// Mitsubishi GX Works2 project: FinalProject   PLC: FX3U/FX3UC

// global labels: Global1
VAR_GLOBAL
  Pos_RedArea AT D109 : INT;
  Pos_AreaA AT D110 : INT;
  End_Home AT M300 : BOOL;
  End_Prepare AT M301 : BOOL;
  Move_Home AT M329 : BOOL;
  En_GetA AT M303 : BOOL;
  GetA AT M304 : BOOL;
  En_GoRed AT M305 : BOOL;
  Go_Red AT M306 : BOOL;
  En_GoBlue AT M307 : BOOL;
  GoBlue AT M308 : BOOL;
  En_Go_A AT M309 : BOOL;
  Go_A AT M310 : BOOL;
  En_Go_B AT M311 : BOOL;
  Go_B AT M312 : BOOL;
  En_GetB AT M313 : BOOL;
  GetB AT M314 : BOOL;
  M_Dem AT M315 : BOOL;
  End_Arr_Red AT M317 : BOOL;
  M_timer AT M318 : BOOL;
  Start_Home AT M319 : BOOL;
  End_ComeBack AT M320 : BOOL;
  Start_B AT X003 : BOOL;
  Stop_B AT X004 : BOOL;
  Emer_B AT M323 : BOOL;
  Go_Home AT M324 : BOOL;
  END_GOHOME AT M325 : BOOL;
  end_get_ProA AT M326 : BOOL;
  M_Xoay AT M327 : BOOL;
  End_RedArea AT M328 : BOOL;
  M_T1 AT M330 : BOOL;
  M_Arr AT M331 : BOOL;
  M_T2 AT M332 : BOOL;
  M_T3 AT M333 : BOOL;
  M_T7 AT M334 : BOOL;
  M_ComeBack AT M335 : BOOL;
  End_Finish AT M336 : BOOL;
  M_T5 AT M337 : BOOL;
  M_Prepare AT S338 : BOOL;
  M_Start AT M321 : BOOL;
  M_Stop AT M322 : BOOL;
END_VAR

PROGRAM MAIN
VAR
  Move_Data_1 : Move_Data;
END_VAR
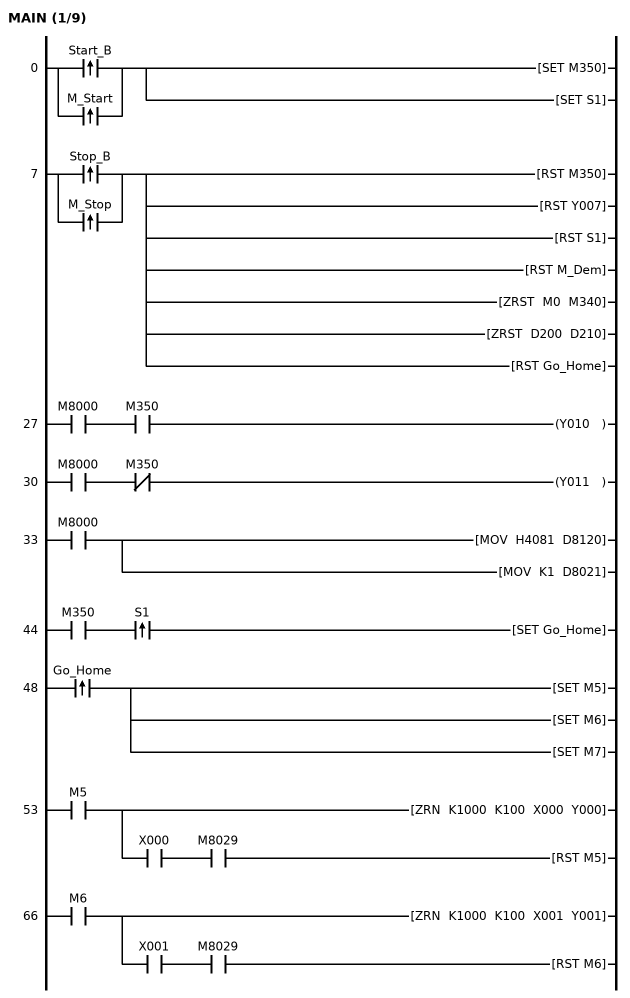
0     LDP     Start_B
      ORP     M_Start
      SET     M350
      SET     S1
7     LDP     Stop_B
      ORP     M_Stop
      RST     M350
      RST     Y007
      RST     S1
      RST     M_Dem
      ZRST    M0 M340
      ZRST    D200 D210
      RST     Go_Home
27    LD      M8000
      AND     M350
      OUT     Y010
30    LD      M8000
      ANI     M350
      OUT     Y011
33    LD      M8000
      MOV     H4081 D8120
      MOV     K1 D8021
44    LD      M350
      ANDP    S1
      SET     Go_Home
48    LDP     Go_Home
      SET     M5
      SET     M6
      SET     M7
53    LD      M5
      ZRN     K1000 K100 X000 Y000
      AND     X000
      AND     M8029
      RST     M5
66    LD      M6
      ZRN     K1000 K100 X001 Y001
      AND     X001
      AND     M8029
      RST     M6
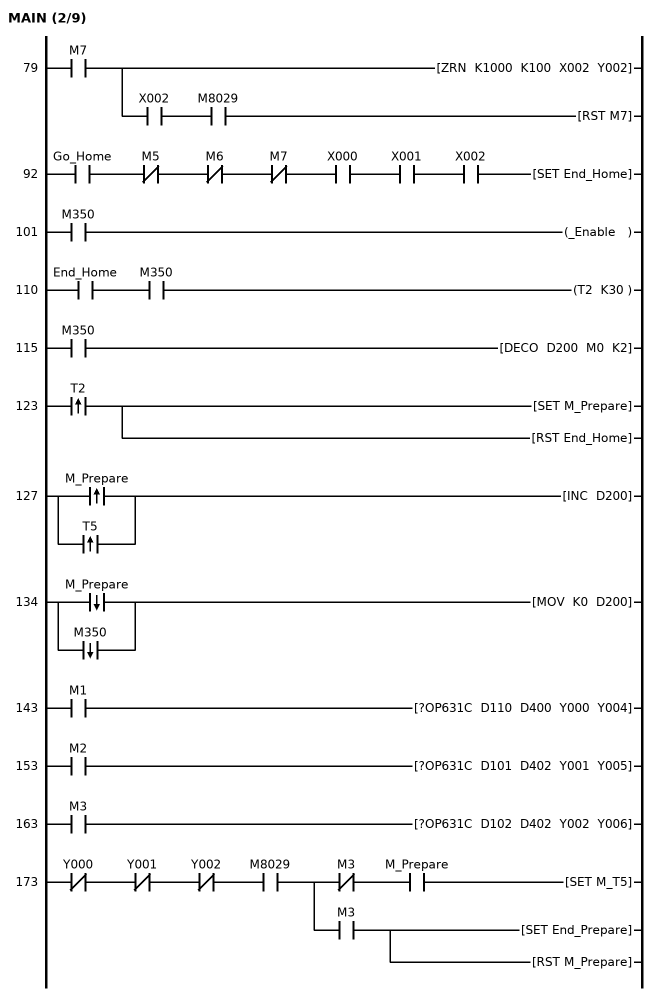
79    LD      M7
      ZRN     K1000 K100 X002 Y002
      AND     X002
      AND     M8029
      RST     M7
92    LD      Go_Home
      ANI     M5
      ANI     M6
      ANI     M7
      AND     X000
      AND     X001
      AND     X002
      SET     End_Home
; FB BLK START Move_Data(Move_Data_1)
101   LD      M350
      OUT     _Enable
; FB START
; FB_NAME Move_Data
; INSTANCE_NAME Move_Data_1
; FB IN_B:Enable
; FB OUT_Enable:B
; FB END
; FB BLK END
110   LD      End_Home
      AND     M350
      OUT     T2 K30
115   LD      M350
      DECO    D200 M0 K2
123   LDP     T2
      SET     M_Prepare
      RST     End_Home
127   LDP     M_Prepare
      ORP     T5
      INC     D200
134   LDF     M_Prepare
      ORF     M350
      MOV     K0 D200
143   LD      M1
      ?OP631C D110 D400 Y000 Y004
153   LD      M2
      ?OP631C D101 D402 Y001 Y005
163   LD      M3
      ?OP631C D102 D402 Y002 Y006
173   LDI     Y000
      ANI     Y001
      ANI     Y002
      AND     M8029
      MPS
      ANI     M3
      AND     M_Prepare
      SET     M_T5
      MPP
      AND     M3
      SET     End_Prepare
      RST     M_Prepare
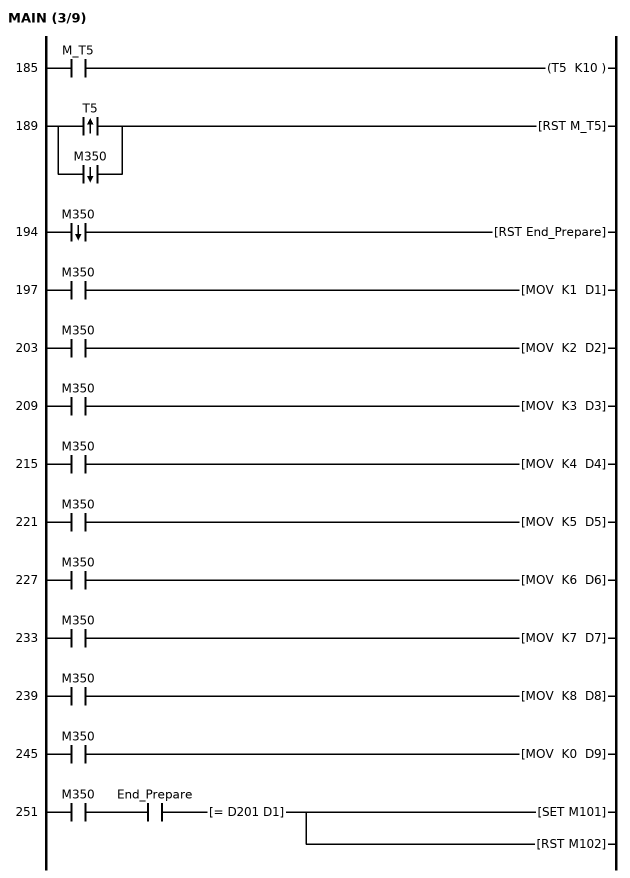
185   LD      M_T5
      OUT     T5 K10
189   LDP     T5
      ORF     M350
      RST     M_T5
194   LDF     M350
      RST     End_Prepare
197   LD      M350
      MOV     K1 D1
203   LD      M350
      MOV     K2 D2
209   LD      M350
      MOV     K3 D3
215   LD      M350
      MOV     K4 D4
221   LD      M350
      MOV     K5 D5
227   LD      M350
      MOV     K6 D6
233   LD      M350
      MOV     K7 D7
239   LD      M350
      MOV     K8 D8
245   LD      M350
      MOV     K0 D9
251   LD      M350
      AND     End_Prepare
      AND=    D201 D1
      SET     M101
      RST     M102
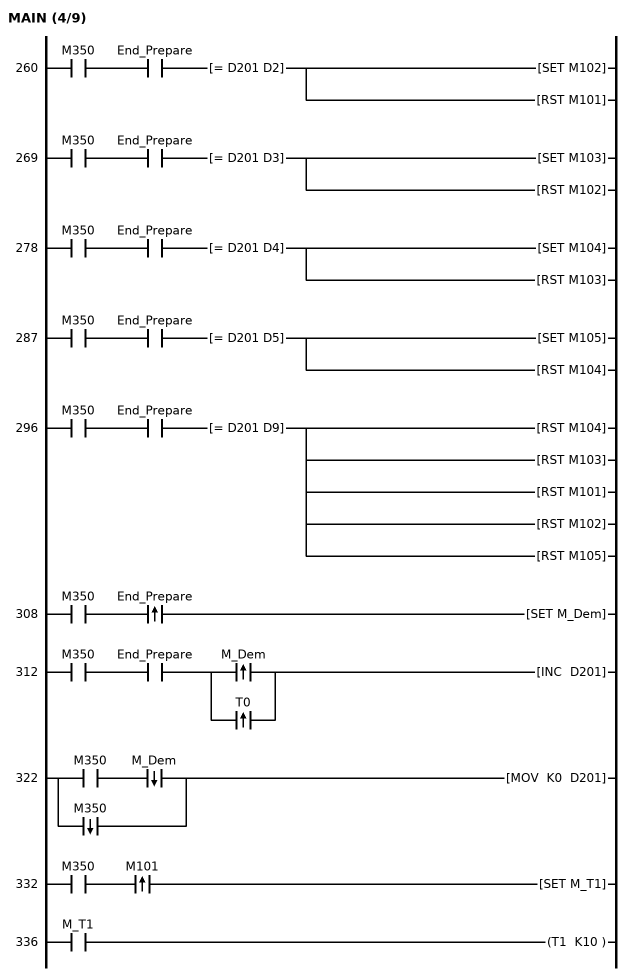
260   LD      M350
      AND     End_Prepare
      AND=    D201 D2
      SET     M102
      RST     M101
269   LD      M350
      AND     End_Prepare
      AND=    D201 D3
      SET     M103
      RST     M102
278   LD      M350
      AND     End_Prepare
      AND=    D201 D4
      SET     M104
      RST     M103
287   LD      M350
      AND     End_Prepare
      AND=    D201 D5
      SET     M105
      RST     M104
296   LD      M350
      AND     End_Prepare
      AND=    D201 D9
      RST     M104
      RST     M103
      RST     M101
      RST     M102
      RST     M105
308   LD      M350
      ANDP    End_Prepare
      SET     M_Dem
312   LD      M350
      AND     End_Prepare
      LDP     M_Dem
      ORP     T0
      ANB
      INC     D201
322   LD      M350
      ANDF    M_Dem
      ORF     M350
      MOV     K0 D201
332   LD      M350
      ANDP    M101
      SET     M_T1
336   LD      M_T1
      OUT     T1 K10
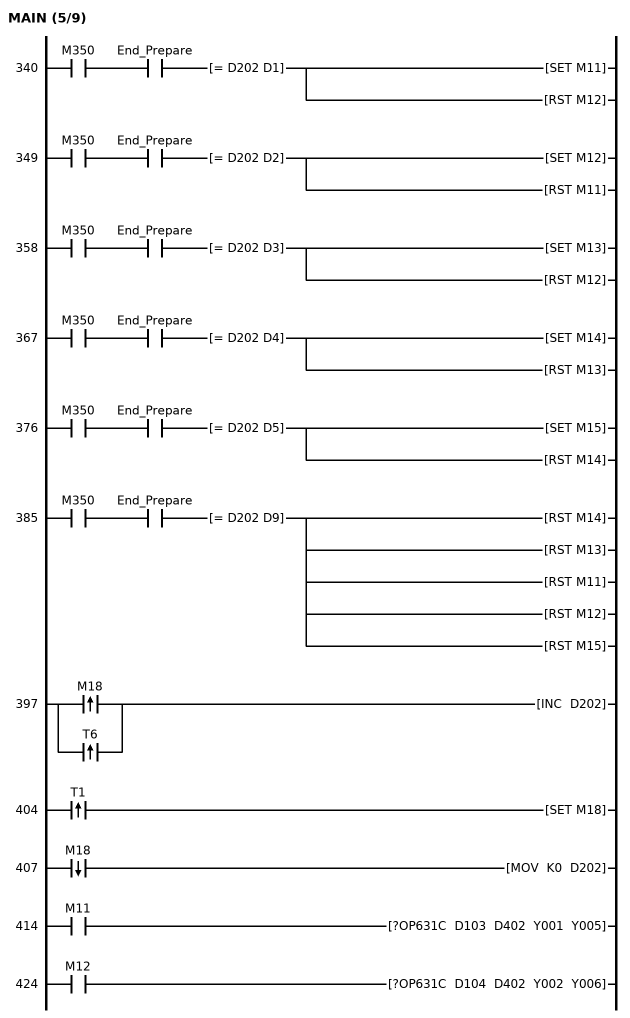
340   LD      M350
      AND     End_Prepare
      AND=    D202 D1
      SET     M11
      RST     M12
349   LD      M350
      AND     End_Prepare
      AND=    D202 D2
      SET     M12
      RST     M11
358   LD      M350
      AND     End_Prepare
      AND=    D202 D3
      SET     M13
      RST     M12
367   LD      M350
      AND     End_Prepare
      AND=    D202 D4
      SET     M14
      RST     M13
376   LD      M350
      AND     End_Prepare
      AND=    D202 D5
      SET     M15
      RST     M14
385   LD      M350
      AND     End_Prepare
      AND=    D202 D9
      RST     M14
      RST     M13
      RST     M11
      RST     M12
      RST     M15
397   LDP     M18
      ORP     T6
      INC     D202
404   LDP     T1
      SET     M18
407   LDF     M18
      MOV     K0 D202
414   LD      M11
      ?OP631C D103 D402 Y001 Y005
424   LD      M12
      ?OP631C D104 D402 Y002 Y006
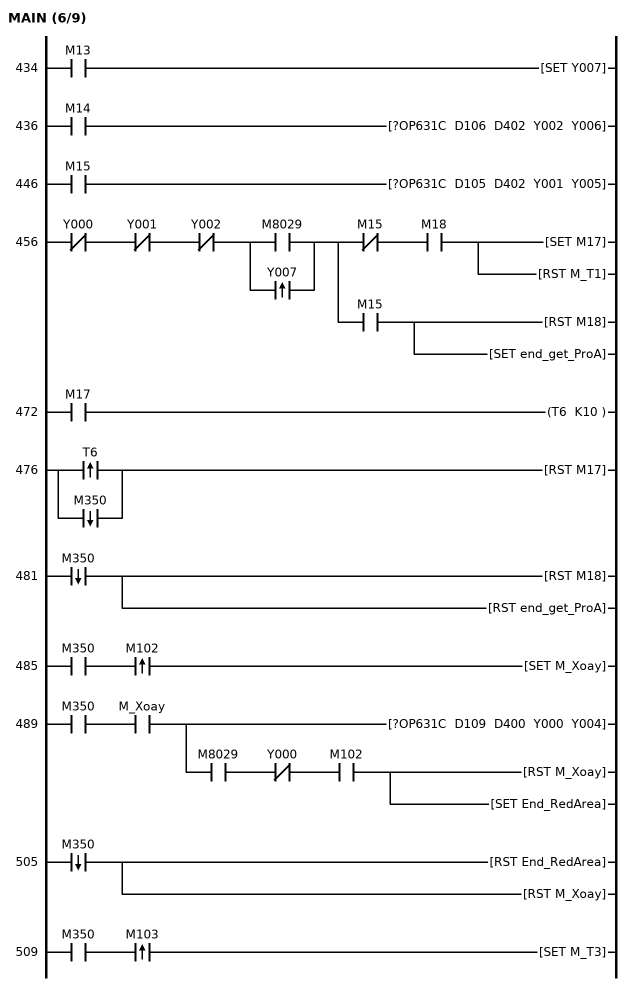
434   LD      M13
      SET     Y007
436   LD      M14
      ?OP631C D106 D402 Y002 Y006
446   LD      M15
      ?OP631C D105 D402 Y001 Y005
456   LDI     Y000
      ANI     Y001
      ANI     Y002
      LD      M8029
      ORP     Y007
      ANB
      MPS
      ANI     M15
      AND     M18
      SET     M17
      RST     M_T1
      MPP
      AND     M15
      RST     M18
      SET     end_get_ProA
472   LD      M17
      OUT     T6 K10
476   LDP     T6
      ORF     M350
      RST     M17
481   LDF     M350
      RST     M18
      RST     end_get_ProA
485   LD      M350
      ANDP    M102
      SET     M_Xoay
489   LD      M350
      AND     M_Xoay
      ?OP631C D109 D400 Y000 Y004
      AND     M8029
      ANI     Y000
      AND     M102
      RST     M_Xoay
      SET     End_RedArea
505   LDF     M350
      RST     End_RedArea
      RST     M_Xoay
509   LD      M350
      ANDP    M103
      SET     M_T3
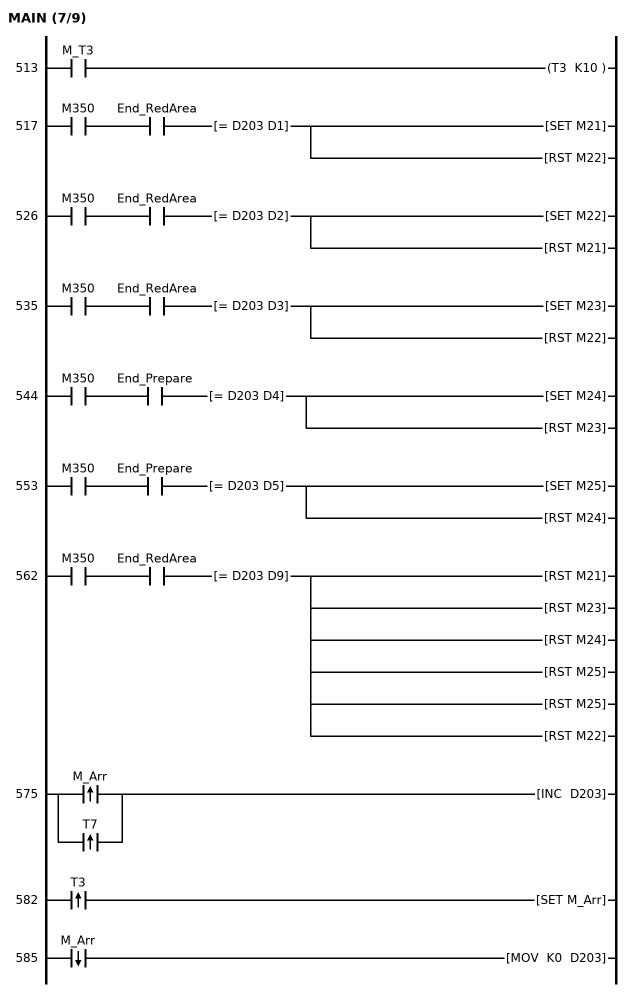
513   LD      M_T3
      OUT     T3 K10
517   LD      M350
      AND     End_RedArea
      AND=    D203 D1
      SET     M21
      RST     M22
526   LD      M350
      AND     End_RedArea
      AND=    D203 D2
      SET     M22
      RST     M21
535   LD      M350
      AND     End_RedArea
      AND=    D203 D3
      SET     M23
      RST     M22
544   LD      M350
      AND     End_Prepare
      AND=    D203 D4
      SET     M24
      RST     M23
553   LD      M350
      AND     End_Prepare
      AND=    D203 D5
      SET     M25
      RST     M24
562   LD      M350
      AND     End_RedArea
      AND=    D203 D9
      RST     M21
      RST     M23
      RST     M24
      RST     M25
      RST     M25
      RST     M22
575   LDP     M_Arr
      ORP     T7
      INC     D203
582   LDP     T3
      SET     M_Arr
585   LDF     M_Arr
      MOV     K0 D203
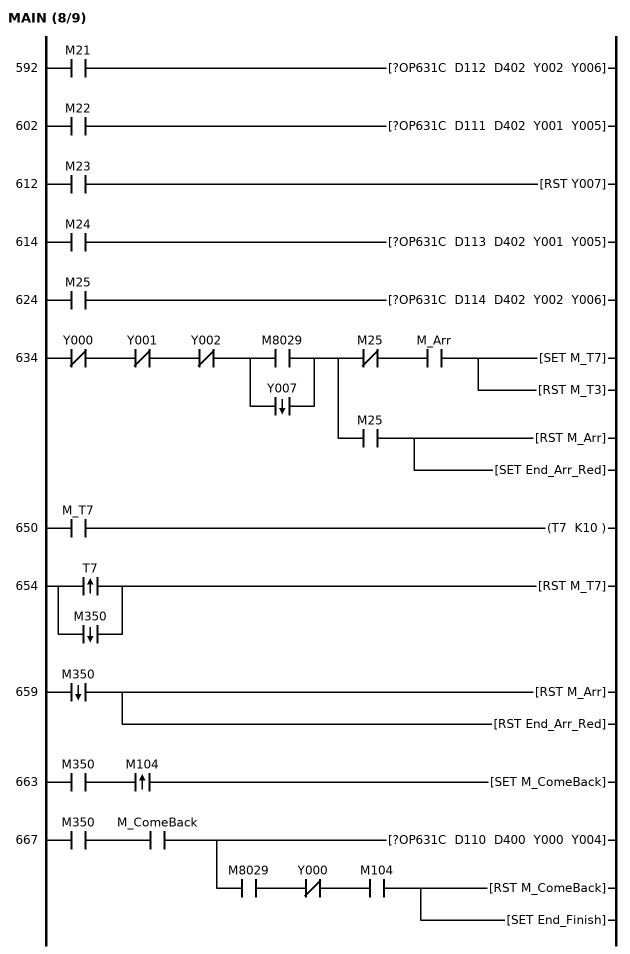
592   LD      M21
      ?OP631C D112 D402 Y002 Y006
602   LD      M22
      ?OP631C D111 D402 Y001 Y005
612   LD      M23
      RST     Y007
614   LD      M24
      ?OP631C D113 D402 Y001 Y005
624   LD      M25
      ?OP631C D114 D402 Y002 Y006
634   LDI     Y000
      ANI     Y001
      ANI     Y002
      LD      M8029
      ORF     Y007
      ANB
      MPS
      ANI     M25
      AND     M_Arr
      SET     M_T7
      RST     M_T3
      MPP
      AND     M25
      RST     M_Arr
      SET     End_Arr_Red
650   LD      M_T7
      OUT     T7 K10
654   LDP     T7
      ORF     M350
      RST     M_T7
659   LDF     M350
      RST     M_Arr
      RST     End_Arr_Red
663   LD      M350
      ANDP    M104
      SET     M_ComeBack
667   LD      M350
      AND     M_ComeBack
      ?OP631C D110 D400 Y000 Y004
      AND     M8029
      ANI     Y000
      AND     M104
      RST     M_ComeBack
      SET     End_Finish
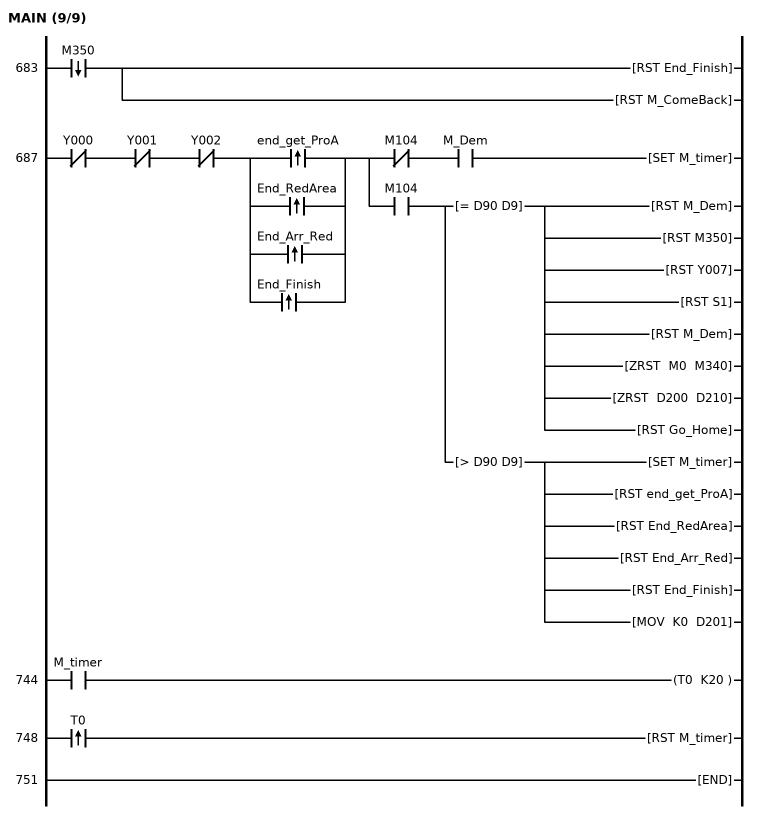
683   LDF     M350
      RST     End_Finish
      RST     M_ComeBack
687   LDI     Y000
      ANI     Y001
      ANI     Y002
      LDP     end_get_ProA
      ORP     End_RedArea
      ORP     End_Arr_Red
      ORP     End_Finish
      ANB
      MPS
      ANI     M104
      AND     M_Dem
      SET     M_timer
      MPP
      AND     M104
      MPS
      AND=    D90 D9
      RST     M_Dem
      RST     M350
      RST     Y007
      RST     S1
      RST     M_Dem
      ZRST    M0 M340
      ZRST    D200 D210
      RST     Go_Home
      MPP
      AND>    D90 D9
      SET     M_timer
      RST     end_get_ProA
      RST     End_RedArea
      RST     End_Arr_Red
      RST     End_Finish
      MOV     K0 D201
744   LD      M_timer
      OUT     T0 K20
748   LDP     T0
      RST     M_timer
751   END
END_PROGRAM

FUNCTION_BLOCK Move_Data
VAR_IN_OUT
  Enable : BOOL;
END_VAR
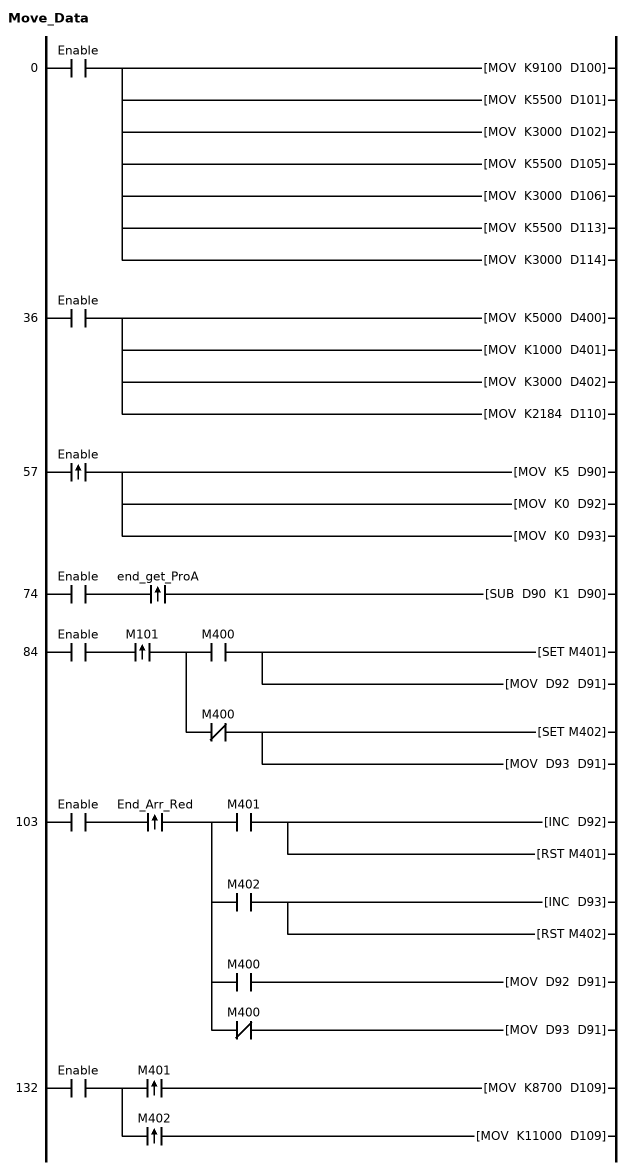
0     LD      Enable
      MOV     K9100 D100
      MOV     K5500 D101
      MOV     K3000 D102
      MOV     K5500 D105
      MOV     K3000 D106
      MOV     K5500 D113
      MOV     K3000 D114
36    LD      Enable
      MOV     K5000 D400
      MOV     K1000 D401
      MOV     K3000 D402
      MOV     K2184 D110
57    LDP     Enable
      MOV     K5 D90
      MOV     K0 D92
      MOV     K0 D93
74    LD      Enable
      ANDP    end_get_ProA
      SUB     D90 K1 D90
84    LD      Enable
      ANDP    M101
      MPS
      AND     M400
      SET     M401
      MOV     D92 D91
      MPP
      ANI     M400
      SET     M402
      MOV     D93 D91
103   LD      Enable
      ANDP    End_Arr_Red
      MPS
      AND     M401
      INC     D92
      RST     M401
      MRD
      AND     M402
      INC     D93
      RST     M402
      MRD
      AND     M400
      MOV     D92 D91
      MPP
      ANI     M400
      MOV     D93 D91
132   LD      Enable
      MPS
      ANDP    M401
      MOV     K8700 D109
      MPP
      ANDP    M402
      MOV     K11000 D109
END_FUNCTION_BLOCK
